FUNCTION_BLOCK EL4132
VAR
	_io : EL4xx2_Data;
	{attribute addProperty Name "WcState"}
	_wcState : WcStateBase;
	{attribute addProperty Name "Info data"}
	_infoData : InfoDataAds;
END_VAR

PROPERTY IO : REFERENCE TO EL4xx2_Data
GET
IO REF= _io;
END_GET
END_PROPERTY

PROPERTY WcState : REFERENCE TO WcStateBase
GET
WcState REF= _wcState;
END_GET
END_PROPERTY

END_FUNCTION_BLOCK

(* stored: Version 1.1.0.1, ProductVersion 3.1.4024.9
   POU EL4132: Id {af29e7ca-ec8e-03b5-0353-b4d8aea9de07}, SpecialFunc None
   Property IO: Id {803f0279-6366-038f-1c5c-3832470c896a}
   Get Get: Id {7c34a465-40d5-07af-11b8-6e988079bd1c}
   Property WcState: Id {c30af17a-082d-0ee8-3c03-709636ba4b58}
   Get Get: Id {0f315138-6db1-0dc5-2b72-96801a2afdb5} *)
